{attribute addProperty BoxType "EL3101-0000-0018"}
{attribute addProperty Id "AI_StandardAT %I*AI_Standard_087F71C73240WcStateAT %I*WcState_F855686C1620InfoDataAT %I*InfoData_BC63D37F80100"}
{attribute addProperty CRC "1089245502"}
{attribute addProperty SizeInBites "128"}
{attribute addProperty SizeInBytes "16"}
TYPE EL3101_60464DCF :
STRUCT
	{attribute addProperty Name "AI_Standard"}
	AI_Standard : AI_Standard_087F71C7;
	{attribute addProperty Name "WcState"}
	WcState : WcState_F855686C;
	{attribute addProperty Name "InfoData"}
	InfoData : InfoData_BC63D37F;
END_STRUCT
END_TYPE

(* stored: Version 1.2.0.0, ProductVersion 3.1.4024.9
   DUT EL3101_60464DCF: Id {82ecc755-a90a-41ee-9583-b0c11f01753a} *)
